{attribute 'qualified_only'}
{attribute 'strict'}
TYPE eDataEntityInvokeType : (
    InvokeAndWaitDone := 0,
    InvokeOnly	 := 10
);
END_TYPE

(* stored: Version 1.1.0.1
   DUT eDataEntityInvokeType: Id {5976a2e1-62c6-0ff6-0696-6562e566c430} *)
